FUNCTION_BLOCK FB_OperatingCounter
VAR_INPUT
	stateString : STRING;
	currentTool : INT;
	SpindleIsOn : BOOL;
END_VAR
VAR_OUTPUT
END_VAR
VAR
	// Timer to count operating time
    runTimer : TON; // Timer On-Delay
    elapsedTime : TIME := T#0S; // Time elapsed since last increment

    // Time interval for incrementing operating hours (e.g., every second)
    timeInterval : TIME := T#1S;

    totalRunHoursRounded : INT;
	totalSawbladeHoursRounded : INT;
	totalHalfInchHoursRounded : INT;
	totalQuarterInchHoursRounded : INT;
END_VAR

totalRunHoursRounded := REAL_TO_INT(GVL_OperationCounter.totalRunHours);
totalSawbladeHoursRounded := REAL_TO_INT(GVL_OperationCounter.totalSawBladeHoursSinceChanged);
totalHalfInchHoursRounded := REAL_TO_INT(GVL_OperationCounter.totalHalfInchHoursSinceChanged);
totalQuarterInchHoursRounded := REAL_TO_INT(GVL_OperationCounter.totalQuarterInchHoursSinceChanged);

IF stateString = 'RUN' OR stateString = 'TOOLCHANGERUN' OR stateString = 'TOOLCHANGEINIT' THEN
	// Timer setup
	runTimer(IN := TRUE, PT := timeInterval);
	elapsedTime := runTimer.ET;
	
	// Check if the timer has elapsed
	IF runTimer.Q THEN
		// Increment operating hours (timeInterval is in seconds, convert to hours)
		GVL_OperationCounter.totalRunHours := GVL_OperationCounter.totalRunHours + TIME_TO_REAL(elapsedTime) / 3600000.0;
		IF SpindleIsOn THEN
			IF currentTool = 0 THEN
				GVL_OperationCounter.totalSawBladeHoursSinceChanged := GVL_OperationCounter.totalSawBladeHoursSinceChanged + TIME_TO_REAL(elapsedTime) / 3600000.0;
			ELSIF currenttool = 2 THEN
				GVL_OperationCounter.totalQuarterInchHoursSinceChanged := GVL_OperationCounter.totalQuarterInchHoursSinceChanged + TIME_TO_REAL(elapsedTime) / 3600000.0;
			ELSIF currenttool = 4 THEN
				GVL_OperationCounter.totalHalfInchHoursSinceChanged := GVL_OperationCounter.totalHalfInchHoursSinceChanged + TIME_TO_REAL(elapsedTime) / 3600000.0;
			END_IF
		END_IF
		// Reset timer
		runTimer(IN := FALSE);
		runTimer(IN := TRUE);
	END_IF
END_IF

END_FUNCTION_BLOCK

(* stored: Version 1.1.0.1, ProductVersion 3.1.4024.12
   POU FB_OperatingCounter: Id {343a864b-43d4-4be9-b0a5-e74d13e6b874}, SpecialFunc None *)
